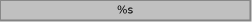
VISUALIZATION V_RadioButton  // 252x22
VAR_INPUT
	IN_Title		: STRING;
	IN_iValue		: INT;
END_VAR
VAR_IN_OUT
	IO_iVar 		: INT;
END_VAR
    Rectangle (0,0 250x20), "%s", text variable: IN_Title, colour toggle: IO_iVar = IN_iValue
        OnMouseClick: execute { IO_iVar := IN_iValue; }
END_VISUALIZATION

(* stored: Version 1.1.0.1, ProductVersion 3.1.4018.10
   Visu V_RadioButton: Id {48c887ea-0db2-4d2c-a7df-c71bd5edee13} *)
